FUNCTION_BLOCK BooleanExpressionFunctionsTest EXTENDS TcUnit.FB_TestSuite

And234();
Or234();
Xor234();

METHOD And234 : BOOL
VAR
	bool1 : BOOL;
	bool2 : BOOL;
	bool3 : BOOL;
	bool4 : BOOL;
	value2 : BoolValue;
	value3 : BoolValue;
	value4 : BoolValue;
	disposable : Disposable;
END_VAR
TcUnit.TEST('Functions And2, 3, 4');

value2 := And2(Bind(bool1), Bind(bool2));
value3 := And3(Bind(bool1), Bind(bool2), Bind(bool3));
value4 := And4(Bind(bool1), Bind(bool2), Bind(bool3), Bind(bool4));

bool1 := FALSE;
bool2 := FALSE;
bool3 := FALSE;
bool4 := FALSE;

AssertEquals_BOOL(
	Expected := FALSE,
	Actual := value2.Value,
	Message := 'FALSE AND FALSE should be FALSE');
AssertEquals_BOOL(
	Expected := FALSE,
	Actual := value3.Value,
	Message := 'FALSE AND FALSE AND FALSE should be FALSE');
AssertEquals_BOOL(
	Expected := FALSE,
	Actual := value4.Value,
	Message := 'FALSE AND FALSE AND FALSE AND FALSE should be FALSE');

bool1 := TRUE;
bool2 := FALSE;
bool3 := FALSE;
bool4 := FALSE;

AssertEquals_BOOL(
	Expected := FALSE,
	Actual := value2.Value,
	Message := 'TRUE AND FALSE should be FALSE');
AssertEquals_BOOL(
	Expected := FALSE,
	Actual := value3.Value,
	Message := 'TRUE AND FALSE AND FALSE should be FALSE');
AssertEquals_BOOL(
	Expected := FALSE,
	Actual := value4.Value,
	Message := 'TRUE AND FALSE AND FALSE AND FALSE should be FALSE');

bool1 := TRUE;
bool2 := TRUE;
bool3 := TRUE;
bool4 := TRUE;

AssertEquals_BOOL(
	Expected := TRUE,
	Actual := value2.Value,
	Message := 'TRUE AND TRUE should be TRUE');
AssertEquals_BOOL(
	Expected := TRUE,
	Actual := value3.Value,
	Message := 'TRUE AND TRUE AND TRUE should be TRUE');
AssertEquals_BOOL(
	Expected := TRUE,
	Actual := value4.Value,
	Message := 'TRUE AND TRUE AND TRUE AND TRUE should be TRUE');

__QUERYINTERFACE(value2, disposable);
disposable.Dispose();
__QUERYINTERFACE(value3, disposable);
disposable.Dispose();
__QUERYINTERFACE(value4, disposable);
disposable.Dispose();

TEST_FINISHED();
END_METHOD

METHOD Or234 : BOOL
VAR
	bool1 : BOOL;
	bool2 : BOOL;
	bool3 : BOOL;
	bool4 : BOOL;
	value2 : BoolValue;
	value3 : BoolValue;
	value4 : BoolValue;
	disposable : Disposable;
END_VAR
TcUnit.TEST('Functions Or2, 3, 4');

value2 := Or2(Bind(bool1), Bind(bool2));
value3 := Or3(Bind(bool1), Bind(bool2), Bind(bool3));
value4 := Or4(Bind(bool1), Bind(bool2), Bind(bool3), Bind(bool4));

bool1 := FALSE;
bool2 := FALSE;
bool3 := FALSE;
bool4 := FALSE;

AssertEquals_BOOL(
	Expected := FALSE,
	Actual := value2.Value,
	Message := 'FALSE OR FALSE should be FALSE');
AssertEquals_BOOL(
	Expected := FALSE,
	Actual := value3.Value,
	Message := 'FALSE OR FALSE OR FALSE should be FALSE');
AssertEquals_BOOL(
	Expected := FALSE,
	Actual := value4.Value,
	Message := 'FALSE OR FALSE OR FALSE OR FALSE should be FALSE');

bool1 := TRUE;
bool2 := FALSE;
bool3 := FALSE;
bool4 := FALSE;

AssertEquals_BOOL(
	Expected := TRUE,
	Actual := value2.Value,
	Message := 'TRUE OR FALSE should be TRUE');
AssertEquals_BOOL(
	Expected := TRUE,
	Actual := value3.Value,
	Message := 'TRUE OR FALSE OR FALSE should be TRUE');
AssertEquals_BOOL(
	Expected := TRUE,
	Actual := value4.Value,
	Message := 'TRUE OR FALSE OR FALSE OR FALSE should be TRUE');

bool1 := TRUE;
bool2 := TRUE;
bool3 := TRUE;
bool4 := TRUE;

AssertEquals_BOOL(
	Expected := TRUE,
	Actual := value2.Value,
	Message := 'TRUE OR TRUE should be TRUE');
AssertEquals_BOOL(
	Expected := TRUE,
	Actual := value3.Value,
	Message := 'TRUE OR TRUE OR TRUE should be TRUE');
AssertEquals_BOOL(
	Expected := TRUE,
	Actual := value4.Value,
	Message := 'TRUE OR TRUE OR TRUE OR TRUE should be TRUE');

__QUERYINTERFACE(value2, disposable);
disposable.Dispose();
__QUERYINTERFACE(value3, disposable);
disposable.Dispose();
__QUERYINTERFACE(value4, disposable);
disposable.Dispose();

TEST_FINISHED();
END_METHOD

METHOD Xor234 : BOOL
VAR
	bool1 : BOOL;
	bool2 : BOOL;
	bool3 : BOOL;
	bool4 : BOOL;
	value2 : BoolValue;
	value3 : BoolValue;
	value4 : BoolValue;
	disposable : Disposable;
END_VAR
TcUnit.TEST('Functions Xor2, 3, 4');

value2 := Xor2(Bind(bool1), Bind(bool2));
value3 := Xor3(Bind(bool1), Bind(bool2), Bind(bool3));
value4 := Xor4(Bind(bool1), Bind(bool2), Bind(bool3), Bind(bool4));

bool1 := FALSE;
bool2 := FALSE;
bool3 := FALSE;
bool4 := FALSE;

AssertEquals_BOOL(
	Expected := FALSE,
	Actual := value2.Value,
	Message := 'FALSE XOR FALSE should be FALSE');
AssertEquals_BOOL(
	Expected := FALSE,
	Actual := value3.Value,
	Message := 'FALSE XOR FALSE XOR FALSE should be FALSE');
AssertEquals_BOOL(
	Expected := FALSE,
	Actual := value4.Value,
	Message := 'FALSE XOR FALSE XOR FALSE XOR FALSE should be FALSE');

bool1 := TRUE;
bool2 := FALSE;
bool3 := FALSE;
bool4 := FALSE;

AssertEquals_BOOL(
	Expected := TRUE,
	Actual := value2.Value,
	Message := 'TRUE XOR FALSE should be TRUE');
AssertEquals_BOOL(
	Expected := TRUE,
	Actual := value3.Value,
	Message := 'TRUE XOR FALSE XOR FALSE should be TRUE');
AssertEquals_BOOL(
	Expected := TRUE,
	Actual := value4.Value,
	Message := 'TRUE XOR FALSE XOR FALSE XOR FALSE should be TRUE');

bool1 := TRUE;
bool2 := TRUE;
bool3 := TRUE;
bool4 := TRUE;

AssertEquals_BOOL(
	Expected := FALSE,
	Actual := value2.Value,
	Message := 'TRUE XOR TRUE should be FALSE');
AssertEquals_BOOL(
	Expected := TRUE,
	Actual := value3.Value,
	Message := 'TRUE XOR TRUE XOR TRUE should be TRUE');
AssertEquals_BOOL(
	Expected := FALSE,
	Actual := value4.Value,
	Message := 'TRUE XOR TRUE XOR TRUE XOR TRUE should be FALSE');

__QUERYINTERFACE(value2, disposable);
disposable.Dispose();
__QUERYINTERFACE(value3, disposable);
disposable.Dispose();
__QUERYINTERFACE(value4, disposable);
disposable.Dispose();

TEST_FINISHED();
END_METHOD

END_FUNCTION_BLOCK

(* stored: Version 1.1.0.1, ProductVersion 3.1.4024.12
   POU BooleanExpressionFunctionsTest: Id {08c31312-6fc2-0947-20dd-b3a488df2c89}, SpecialFunc None
   Method And234: Id {7430b17d-5618-0534-3882-c682b0e33d85}
   Method Or234: Id {75613706-43c7-070c-3e1f-e775bccf9d25}
   Method Xor234: Id {a53167e1-fcec-0820-2994-53437c59f319} *)
